{attribute 'GeneratedUsingTerminal: EK1110-0000-0017'}
{attribute addProperty BoxType "EK1110-0000-0017"}
{attribute addProperty Description "EK1110 EtherCAT extension"}
{attribute addProperty Physics "KY"}
{attribute addProperty Id "InfoDataAT %I*InfoData_6F19DB2B2"}
{attribute addProperty CRC "532711307"}
{attribute addProperty Size "2"}
TYPE EK1110_1FC0878B EXTENDS TcoIo.EtcSlaveTerminalBase_947E5A46 :
STRUCT
	{attribute addProperty Name "InfoData"}
	InfoData : TcoIo.InfoData_6F19DB2B;
END_STRUCT
END_TYPE

(* stored: Version 1.2.0.0, ProductVersion 3.1.4024.11
   DUT EK1110_1FC0878B: Id {30f0d2e5-f3b9-03e3-1835-1e9000fcb585} *)
